(* CODESYS project 30_powerflex_speed_label_wide.export

Project tree, tasks and I/O mapping:
  Device : CODESYS Control Win V3 x64, CODESYS, version 3.5.22.20
    application Application
      libraries: VisuDialogs, * (System)
      task MainTask (cyclic, interval t#20ms, priority 1) calls PLC_PRG
      task VISU_TASK (cyclic, interval 100 ms, priority 31) calls VisuElems.Visu_Prg
      program PLC_PRG [ST]
      function block TF_PowerFlex525_Core [ST]
      visualisation VISU_PowerFlex525_Test
*)

// Device/Application/PLC_PRG
PROGRAM PLC_PRG
VAR
	fbPowerFlex525: TF_PowerFlex525_Core;
	diInp_Source: DINT;
	xInp_PRunFwd: BOOL;
	xInp_PRunRev: BOOL;
	xInp_PJogFwd: BOOL;
	xInp_PJogRev: BOOL;
	xInp_PStop: BOOL;
	xInp_PReset: BOOL;
	rInp_PSpeed: REAL;
	xInp_ORunFwd: BOOL;
	xInp_ORunRev: BOOL;
	xInp_OJogFwd: BOOL;
	xInp_OJogRev: BOOL;
	xInp_OStop: BOOL;
	xInp_OReset: BOOL;
	rInp_OSpeed: REAL;
	xInp_XRunFwd: BOOL;
	xInp_XRunRev: BOOL;
	xInp_XJogFwd: BOOL;
	xInp_XJogRev: BOOL;
	xInp_XStop: BOOL;
	xInp_XReset: BOOL;
	rInp_XSpeed: REAL;
	xInp_MRunFwd: BOOL;
	xInp_MRunRev: BOOL;
	xInp_MJogFwd: BOOL;
	xInp_MJogRev: BOOL;
	xInp_MStop: BOOL;
	xInp_MReset: BOOL;
	rInp_MSpeed: REAL;
	diInp_OvCmd: DINT;
	rInp_OvSpeed: REAL;
	xInp_PSetOverride: BOOL;
	rInp_MPSet: REAL;
	xInp_PermOK: BOOL;
	xInp_NBPermOK: BOOL;
	xInp_IntlkOK: BOOL;
	xInp_NBIntlkOK: BOOL;
	xInp_Bypass: BOOL;
	xInp_RunFwdAvail: BOOL;
	xInp_RunRevAvail: BOOL;
	xInp_JogFwdAvail: BOOL;
	xInp_JogRevAvail: BOOL;
	xInp_Ready: BOOL;
	xInp_Active: BOOL;
	xInp_ENetLogicCtrl: BOOL;
	xInp_KeypadCtrlSts: BOOL;
	xInp_KeypadCtrlCmd: BOOL;
	rInp_MaxSpeed: REAL;
	rInp_JogSpeed: REAL;
	diInp_StartDelayMs: DINT;
	diInp_ElapsedMs: DINT;
	uiOut_LogicCommand: UINT;
	iOut_SpeedCommand: INT;
	rOut_RefSpeed: REAL;
	xOut_PermOK: BOOL;
	xOut_IntlkOK: BOOL;
	xOut_RunFwd: BOOL;
	xOut_RunRev: BOOL;
	xOut_JogFwd: BOOL;
	xOut_JogRev: BOOL;
	xOut_Starting: BOOL;
	xOut_Stopping: BOOL;
END_VAR

fbPowerFlex525(
    Inp_Source := diInp_Source,
    Inp_PRunFwd := xInp_PRunFwd,
    Inp_PRunRev := xInp_PRunRev,
    Inp_PJogFwd := xInp_PJogFwd,
    Inp_PJogRev := xInp_PJogRev,
    Inp_PStop := xInp_PStop,
    Inp_PReset := xInp_PReset,
    Inp_PSpeed := rInp_PSpeed,
    Inp_ORunFwd := xInp_ORunFwd,
    Inp_ORunRev := xInp_ORunRev,
    Inp_OJogFwd := xInp_OJogFwd,
    Inp_OJogRev := xInp_OJogRev,
    Inp_OStop := xInp_OStop,
    Inp_OReset := xInp_OReset,
    Inp_OSpeed := rInp_OSpeed,
    Inp_XRunFwd := xInp_XRunFwd,
    Inp_XRunRev := xInp_XRunRev,
    Inp_XJogFwd := xInp_XJogFwd,
    Inp_XJogRev := xInp_XJogRev,
    Inp_XStop := xInp_XStop,
    Inp_XReset := xInp_XReset,
    Inp_XSpeed := rInp_XSpeed,
    Inp_MRunFwd := xInp_MRunFwd,
    Inp_MRunRev := xInp_MRunRev,
    Inp_MJogFwd := xInp_MJogFwd,
    Inp_MJogRev := xInp_MJogRev,
    Inp_MStop := xInp_MStop,
    Inp_MReset := xInp_MReset,
    Inp_MSpeed := rInp_MSpeed,
    Inp_OvCmd := diInp_OvCmd,
    Inp_OvSpeed := rInp_OvSpeed,
    Inp_PSetOverride := xInp_PSetOverride,
    Inp_MPSet := rInp_MPSet,
    Inp_PermOK := xInp_PermOK,
    Inp_NBPermOK := xInp_NBPermOK,
    Inp_IntlkOK := xInp_IntlkOK,
    Inp_NBIntlkOK := xInp_NBIntlkOK,
    Inp_Bypass := xInp_Bypass,
    Inp_RunFwdAvail := xInp_RunFwdAvail,
    Inp_RunRevAvail := xInp_RunRevAvail,
    Inp_JogFwdAvail := xInp_JogFwdAvail,
    Inp_JogRevAvail := xInp_JogRevAvail,
    Inp_Ready := xInp_Ready,
    Inp_Active := xInp_Active,
    Inp_ENetLogicCtrl := xInp_ENetLogicCtrl,
    Inp_KeypadCtrlSts := xInp_KeypadCtrlSts,
    Inp_KeypadCtrlCmd := xInp_KeypadCtrlCmd,
    Inp_MaxSpeed := rInp_MaxSpeed,
    Inp_JogSpeed := rInp_JogSpeed,
    Inp_StartDelayMs := diInp_StartDelayMs,
    Inp_ElapsedMs := diInp_ElapsedMs,
    Out_LogicCommand => uiOut_LogicCommand,
    Out_SpeedCommand => iOut_SpeedCommand,
    Out_RefSpeed => rOut_RefSpeed,
    Out_PermOK => xOut_PermOK,
    Out_IntlkOK => xOut_IntlkOK,
    Out_RunFwd => xOut_RunFwd,
    Out_RunRev => xOut_RunRev,
    Out_JogFwd => xOut_JogFwd,
    Out_JogRev => xOut_JogRev,
    Out_Starting => xOut_Starting,
    Out_Stopping => xOut_Stopping
);

END_PROGRAM

// Device/Application/TF_PowerFlex525_Core
FUNCTION_BLOCK TF_PowerFlex525_Core
VAR_INPUT
	Inp_Source: DINT;
	Inp_PRunFwd: BOOL;
	Inp_PRunRev: BOOL;
	Inp_PJogFwd: BOOL;
	Inp_PJogRev: BOOL;
	Inp_PStop: BOOL;
	Inp_PReset: BOOL;
	Inp_PSpeed: REAL;
	Inp_ORunFwd: BOOL;
	Inp_ORunRev: BOOL;
	Inp_OJogFwd: BOOL;
	Inp_OJogRev: BOOL;
	Inp_OStop: BOOL;
	Inp_OReset: BOOL;
	Inp_OSpeed: REAL;
	Inp_XRunFwd: BOOL;
	Inp_XRunRev: BOOL;
	Inp_XJogFwd: BOOL;
	Inp_XJogRev: BOOL;
	Inp_XStop: BOOL;
	Inp_XReset: BOOL;
	Inp_XSpeed: REAL;
	Inp_MRunFwd: BOOL;
	Inp_MRunRev: BOOL;
	Inp_MJogFwd: BOOL;
	Inp_MJogRev: BOOL;
	Inp_MStop: BOOL;
	Inp_MReset: BOOL;
	Inp_MSpeed: REAL;
	Inp_OvCmd: DINT;
	Inp_OvSpeed: REAL;
	Inp_PSetOverride: BOOL;
	Inp_MPSet: REAL;
	Inp_PermOK: BOOL;
	Inp_NBPermOK: BOOL;
	Inp_IntlkOK: BOOL;
	Inp_NBIntlkOK: BOOL;
	Inp_Bypass: BOOL;
	Inp_RunFwdAvail: BOOL;
	Inp_RunRevAvail: BOOL;
	Inp_JogFwdAvail: BOOL;
	Inp_JogRevAvail: BOOL;
	Inp_Ready: BOOL;
	Inp_Active: BOOL;
	Inp_ENetLogicCtrl: BOOL;
	Inp_KeypadCtrlSts: BOOL;
	Inp_KeypadCtrlCmd: BOOL;
	Inp_MaxSpeed: REAL;
	Inp_JogSpeed: REAL;
	Inp_StartDelayMs: DINT;
	Inp_ElapsedMs: DINT;
END_VAR
VAR_OUTPUT
	Out_LogicCommand: UINT;
	Out_SpeedCommand: INT;
	Out_RefSpeed: REAL;
	Out_PermOK: BOOL;
	Out_IntlkOK: BOOL;
	Out_RunFwd: BOOL;
	Out_RunRev: BOOL;
	Out_JogFwd: BOOL;
	Out_JogRev: BOOL;
	Out_Starting: BOOL;
	Out_Stopping: BOOL;
END_VAR
VAR
	RunFwd: BOOL;
	RunRev: BOOL;
	StartElapsedMs: DINT;
	TimerDone: BOOL;
	StopCmd: BOOL;
	StartCmd: BOOL;
	JogCmd: BOOL;
	ResetCmd: BOOL;
	SpeedRef: REAL;
END_VAR

Out_PermOK := ((Inp_PermOK OR Inp_Bypass) AND Inp_NBPermOK);
Out_IntlkOK := ((Inp_IntlkOK OR Inp_Bypass) AND Inp_NBIntlkOK);
IF (Inp_Source = 1) THEN
    IF Inp_PSetOverride THEN
        Out_RefSpeed := Inp_MPSet;
    ELSE
        Out_RefSpeed := Inp_PSpeed;
    END_IF;
    RunFwd := (((Inp_PRunFwd AND (Out_PermOK OR RunFwd)) AND Out_IntlkOK) AND NOT (Inp_PStop));
    RunRev := (((Inp_PRunRev AND (Out_PermOK OR RunRev)) AND Out_IntlkOK) AND NOT (Inp_PStop));
ELSIF (Inp_Source = 2) THEN
    Out_RefSpeed := Inp_OSpeed;
    RunFwd := (((RunFwd OR (((Inp_ORunFwd AND Inp_RunFwdAvail) AND Out_PermOK) AND NOT (Inp_ORunRev))) AND Out_IntlkOK) AND NOT (Inp_OStop));
    RunRev := (((RunRev OR (((Inp_ORunRev AND Inp_RunRevAvail) AND Out_PermOK) AND NOT (Inp_ORunFwd))) AND Out_IntlkOK) AND NOT (Inp_OStop));
ELSIF (Inp_Source = 3) THEN
    Out_RefSpeed := Inp_XSpeed;
    RunFwd := (((RunFwd OR (((Inp_XRunFwd AND Inp_RunFwdAvail) AND Out_PermOK) AND NOT (Inp_XRunRev))) AND Out_IntlkOK) AND NOT (Inp_XStop));
    RunRev := (((RunRev OR (((Inp_XRunRev AND Inp_RunRevAvail) AND Out_PermOK) AND NOT (Inp_XRunFwd))) AND Out_IntlkOK) AND NOT (Inp_XStop));
ELSIF (Inp_Source = 4) THEN
    Out_RefSpeed := Inp_OvSpeed;
    IF ((Inp_OvCmd = 1) OR NOT (Out_IntlkOK)) THEN
        RunFwd := FALSE;
        RunRev := FALSE;
    ELSIF ((Inp_OvCmd = 2) AND Out_PermOK) THEN
        RunRev := FALSE;
        RunFwd := TRUE;
    ELSIF ((Inp_OvCmd = 3) AND Out_PermOK) THEN
        RunFwd := FALSE;
        RunRev := TRUE;
    END_IF;
ELSIF (Inp_Source = 5) THEN
    Out_RefSpeed := Inp_MSpeed;
    RunFwd := (((RunFwd OR (((Inp_MRunFwd AND Inp_RunFwdAvail) AND Out_PermOK) AND NOT (Inp_MRunRev))) AND Out_IntlkOK) AND NOT (Inp_MStop));
    RunRev := (((RunRev OR (((Inp_MRunRev AND Inp_RunRevAvail) AND Out_PermOK) AND NOT (Inp_MRunFwd))) AND Out_IntlkOK) AND NOT (Inp_MStop));
ELSE
    Out_RefSpeed := 0.0;
    RunFwd := FALSE;
    RunRev := FALSE;
END_IF;
Out_JogFwd := (((Inp_JogFwdAvail AND Out_PermOK) AND (((((Inp_Source = 2) AND Inp_OJogFwd) AND NOT (Inp_OJogRev)) OR (((Inp_Source = 3) AND Inp_XJogFwd) AND NOT (Inp_XJogRev))) OR (((Inp_Source = 5) AND Inp_MJogFwd) AND NOT (Inp_MJogRev)))) OR (((Inp_Source = 1) AND Inp_PJogFwd) AND NOT (Inp_PJogRev)));
Out_JogRev := (((Inp_JogRevAvail AND Out_PermOK) AND (((((Inp_Source = 2) AND Inp_OJogRev) AND NOT (Inp_OJogFwd)) OR (((Inp_Source = 3) AND Inp_XJogRev) AND NOT (Inp_XJogFwd))) OR (((Inp_Source = 5) AND Inp_MJogRev) AND NOT (Inp_MJogFwd)))) OR (((Inp_Source = 1) AND Inp_PJogRev) AND NOT (Inp_PJogFwd)));
IF (RunFwd OR RunRev) THEN
    StartElapsedMs := (StartElapsedMs + Inp_ElapsedMs);
    IF (StartElapsedMs >= Inp_StartDelayMs) THEN
        StartElapsedMs := Inp_StartDelayMs;
        TimerDone := TRUE;
    ELSE
        TimerDone := FALSE;
    END_IF;
ELSE
    StartElapsedMs := 0;
    TimerDone := FALSE;
END_IF;
Out_Starting := ((RunFwd OR RunRev) AND NOT (TimerDone));
StopCmd := ((Inp_Active AND Inp_ENetLogicCtrl) AND NOT (((((Inp_KeypadCtrlSts OR RunFwd) OR RunRev) OR Out_JogFwd) OR Out_JogRev)));
StartCmd := (((Inp_Ready AND TimerDone) AND NOT (StopCmd)) AND (((RunFwd OR RunRev) OR Out_JogFwd) OR Out_JogRev));
JogCmd := ((Inp_Ready AND NOT (((StopCmd OR RunFwd) OR RunRev))) AND (Out_JogFwd OR Out_JogRev));
ResetCmd := (((Inp_PReset OR Inp_OReset) OR Inp_XReset) OR Inp_MReset);
Out_LogicCommand := 0;
IF StopCmd THEN
    Out_LogicCommand := (Out_LogicCommand + 1);
END_IF;
IF StartCmd THEN
    Out_LogicCommand := (Out_LogicCommand + 2);
END_IF;
IF JogCmd THEN
    Out_LogicCommand := (Out_LogicCommand + 4);
END_IF;
IF ResetCmd THEN
    Out_LogicCommand := (Out_LogicCommand + 8);
END_IF;
IF (RunFwd OR Out_JogFwd) THEN
    Out_LogicCommand := (Out_LogicCommand + 16);
END_IF;
IF (RunRev OR Out_JogRev) THEN
    Out_LogicCommand := (Out_LogicCommand + 32);
END_IF;
IF Inp_KeypadCtrlCmd THEN
    Out_LogicCommand := (Out_LogicCommand + 64);
END_IF;
IF (Out_JogFwd OR Out_JogRev) THEN
    SpeedRef := Inp_JogSpeed;
ELSE
    SpeedRef := Out_RefSpeed;
END_IF;
IF (SpeedRef < 0.0) THEN
    SpeedRef := 0.0;
ELSIF (SpeedRef > Inp_MaxSpeed) THEN
    SpeedRef := Inp_MaxSpeed;
END_IF;
Out_SpeedCommand := REAL_TO_INT((SpeedRef * 100.0));
Out_RunFwd := RunFwd;
Out_RunRev := RunRev;
Out_Stopping := (Inp_Active AND NOT ((((RunFwd OR RunRev) OR Out_JogFwd) OR Out_JogRev)));

END_FUNCTION_BLOCK

// Device/Application/VISU_PowerFlex525_Test
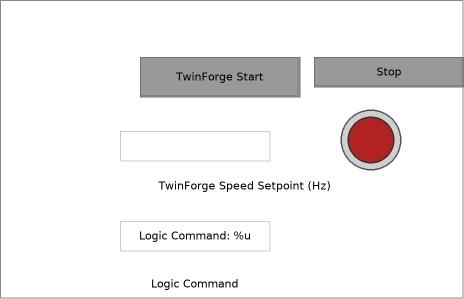
VISUALIZATION VISU_PowerFlex525_Test  // 464x299
    Button (140,57 160x40), "TwinForge Start"
    Button (314,57 150x30), "Stop"
        toggle PLC_PRG.xInp_PStop
    Textfield (120,131 150x30)
        OnMouseClick: write PLC_PRG.rInp_PSpeed via VisuDialogs.Keypad, min 0, max 70, title 'Speed Setpoint (Hz)', format %.1f
    Lamp1 (336,105 70x70), variable: PLC_PRG.xOut_RunFwd, style: Lamp-Lamp1-Red
    Label (120,171 250x30), "TwinForge Speed Setpoint (Hz)"
    Textfield (120,221 150x30), "Logic Command: %u", text variable: PLC_PRG.uiOut_LogicCommand
    Label (120,269 150x30), "Logic Command"
END_VISUALIZATION
